FUNCTION_BLOCK CL_AxisMCL1LeftFront EXTENDS CL_AxisMC
VAR
  objAxisDriver : CL_AxisDriverL1LeftFront;
END_VAR

SUPER^();

METHOD PUBLIC Init : BOOL
VAR_INPUT
  stIrrLine       : ST_LineReference;
  stAxisMotor_P	  : POINTER TO AXIS_REF;
  stAxisMaster_P  : POINTER TO AXIS_REF;
  stDriver        : POINTER TO ST_DriverAX8206_HWI;
END_VAR
Init := FALSE;
IF stDriver <> 0 THEN
  Init := objAxisDriver.Init(stDriver := stDriver);
  Init := Init AND SUPER^.InitMC(stIrrLine := stIrrLine, stAxisMotor_P := stAxisMotor_P, stAxisMaster_P := stAxisMaster_P, AxisDriver_P := ADR(objAxisDriver));
END_IF
END_METHOD

METHOD PROTECTED InitDefect : BOOL
InitDefect := SUPER^.InitDefect();
ADSLOGSTR(ADSLOG_MSGTYPE_LOG, 'CL_AxisMCL1LeftFront init defect','');
END_METHOD

METHOD PROTECTED InitParams : BOOL
VAR_INPUT
END_VAR
InitParams := SUPER^.InitParams();
_sWhichAxis := 'left(L1)-front';
_lrInverse := 1.0;
END_METHOD

END_FUNCTION_BLOCK

(* stored: Version 1.1.0.1, ProductVersion 3.1.4024.12
   POU CL_AxisMCL1LeftFront: Id {d5d457c4-b3f3-4d4e-906d-770cc886d557}, SpecialFunc None
   Method Init: Id {2c8b3418-2026-4837-85f8-34b53282222a}
   Method InitDefect: Id {5b773ca0-6402-4f85-8ced-27749da5bd34}
   Method InitParams: Id {3186c497-859f-49a0-a777-0d308434e9d2} *)
